FUNCTION_BLOCK AE_SWITCH (* Switching (demultiplexing) an event based on boolean input G *)
  (* Standard: 61499-1 Annex A; Description: Copyright (c) 2017 fortiss GmbH This program and the accompanying materials are made available under the terms of the Eclipse Public License 2.0 which is available at https://www.eclipse.org/legal/epl-2.0/ SPDX-License-Identifier: EPL-2.0 *)
  (* Version 3.0, 2025-04-14, Patrick Aigner, changed package *)
  (* Version 1.0, 2017-09-21, Alois Zoitl, fortiss GmbH, initial API and implementation and/or initial documentation *)
  PACKAGE adapter::events::unidirectional;
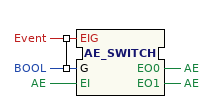
  EVENT_INPUT
    EIG WITH G; (* set G *)
  END_EVENT
  VAR_INPUT
    G : BOOL; (* Switch EI to EO0 when G=0, to EO1 when G=1 *)
  END_VAR
  SOCKETS
    EI : adapter::types::unidirectional::AE; (* Event Input *)
  END_SOCKETS
  PLUGS
    EO0 : adapter::types::unidirectional::AE; (* Output, switched from EI when G=0 *)
    EO1 : adapter::types::unidirectional::AE; (* Output, switched from EI when G=1 *)
  END_PLUGS
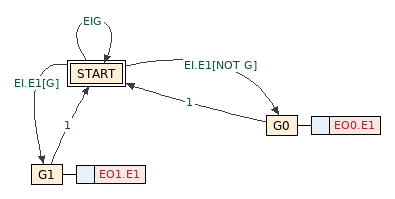
  EC_STATES
    START; (* Initial State *)
    G0 : -> EO0.E1; (* Issue EO0 when EI arrives with G=0 *)
    G1 : -> EO1.E1; (* Issue EO1 when EI arrives with G=1 *)
  END_STATES
  EC_TRANSITIONS
    G0 TO START := 1;
    G1 TO START := 1;
    START TO G0 := EI.E1[NOT G];
    START TO G1 := EI.E1[G];
    START TO START := EIG;
  END_TRANSITIONS
END_FUNCTION_BLOCK
